{attribute 'qualified_only'}
VAR_GLOBAL CONSTANT
	
END_VAR
VAR_GLOBAL
	//
	bAllUnitsReady						: BOOL;					// All machine units are OK, and ready to operate
	bGeneralOK							: BOOL;					// There is no Warning, Error or Fatal Error - just when it's true - You can operate
	bGeneralWarning						: BOOL;					// Warning - just message/event - no reaction
	bGeneralError						: BOOL;					// Error - machine has to stop, start is possible from this position
	bGeneralFatalError					: BOOL;					// Fatal error causes machine stop. You have to go back for cycle begin.

	// 
	bRestartRequired					: BOOL;					// In case of fatal error, when whole process restart required
	bMuteGeneralError					: BOOL;					// Just for service/maitenance - if You are aware of consequences You can force muting mode
	bMuteGeneralFatalError				: BOOL;					// Just for service/maitenance - if You are aware of consequences You can force muting mode
END_VAR

(* stored: Version 1.1.0.1, ProductVersion 3.1.4022.12
   GVL GVL: Id {3898fc2d-91df-4d02-9331-f90e3791f554} *)
